# B&R Automation Studio project PROJEKT_AS_4_11_2_75_X20CP1382
Automation Studio 4.9

## Configuration Config1

CPU X20CP1382, AutomationRuntime D4.83, Build 4.1.2, Vc V4.72.3

### Task classes (Cpu.sw)
```
Cyclic#4:
  Program <- Program.prg
Binaries: udbdef, FWRules, TCData, sysconf, Role, User, iomap, ashwd, asfw, arconfig, ashwac
Libraries: runtime, astime, asieccon
```

### Hardware
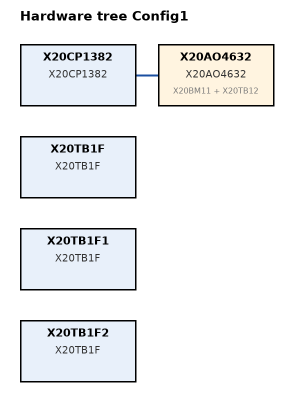
```
X20AO4632 : X20AO4632 v1.2.0.0  [SS1 -> X20TB12.SS; SL -> X20BM11.SL1]
X20BM11 : X20BM11 v1.1.0.0  [X2X1 -> X20CP1382.IF6]
X20CP1382 : X20CP1382 v1.14.0.0  [X1 -> X1.SL; X2 -> X2.SL; X3 -> X3.SL]
  Module X1 (Type=X1, Virtual=true, Version=1.14.0.0)
    Connection (Connector=SS1, TargetModule=X20TB1F, TargetConnector=SS)
    Connection (Connector=SL, TargetModule=X20CP1382, TargetConnector=X1)
  Module X2 (Type=X2, Virtual=true, Version=1.14.0.0)
    Connection (Connector=SS1, TargetModule=X20TB1F1, TargetConnector=SS)
    Connection (Connector=SL, TargetModule=X20CP1382, TargetConnector=X2)
  Module X3 (Type=X3, Virtual=true, Version=1.14.0.0)
    Connection (Connector=SS1, TargetModule=X20TB1F2, TargetConnector=SS)
    Connection (Connector=SL, TargetModule=X20CP1382, TargetConnector=X3)
  Connector IF2:
    ActivateDevice = 1
    Mode = Manual
    InternetAddress = 192.168.10.5
    SubnetMask = 255.255.255.0
    ActivateSnmp = 2
  ConfigurationID = X20CP1382_Config1
  Simulation = 1
X20TB12 : X20TB12 v1.0.0.0
X20TB1F : X20TB1F v1.0.0.0
X20TB1F1 : X20TB1F v1.0.0.0
X20TB1F2 : X20TB1F v1.0.0.0
```

### IoMap.iom - X20CP1382/IoMap.iom
```iecst
VAR_CONFIG
	::Program:speedTreadmill AT %QW."X20AO4632".AnalogOutput01;
	::Program:directionTreadmillright AT %QW."X20AO4632".AnalogOutput02;
	::Program:directionTreadmillleft AT %QW."X20AO4632".AnalogOutput03;
<<<<<<< HEAD
	::Program:Reed_Sensor_Input_1 AT %IW."X1".AnalogInput01;
=======
	::Program:inductiveSensor1_DI AT %IX."X1".DigitalInput01 INVERSE;
	::Program:inductiveSensor2_DI AT %IX."X1".DigitalInput02;
	::Program:peristalticPump1_AO AT %QW."X20AO4632".AnalogOutput04;
>>>>>>> a31492344b22443c312620c2728d9b959337b792
END_VAR
```

## Logical view

### Program Logical/Program

#### Variables.var
```iecst
VAR
	speedTreadmill : INT;
	directionTreadmillleft : INT;
	directionTreadmillright : INT;
<<<<<<< HEAD
	Reed_Sensor_Input_1 : INT;
=======
	inductiveSensor1_DI : BOOL;
	inductiveSensor2_DI : BOOL;
	peristalticPump1_AO : INT;
>>>>>>> a31492344b22443c312620c2728d9b959337b792
END_VAR
```

#### Cyclic.st
```iecst
PROGRAM _CYCLIC
	// IF D11 equals ON -> Power on 10V
	// 32000 = 14,6V
	// 10V =
	speedTreadmill := 30000;
	directionTreadmillleft := 25000;
	//directionTreadmillright := 25000;
	speedTreadmill := -4000;

	peristalticPump1_AO := 10000;
	IF inductiveSensor1_DI = TRUE
	THEN
		directionTreadmillright := 25000;
		directionTreadmillleft := 0;
	ELSIF inductiveSensor2_DI = TRUE THEN
		directionTreadmillleft := 25000;
		directionTreadmillright := 0;
	END_IF;

	//

	//speedTreadmill := -30000;

END_PROGRAM
```

#### Init.st
```iecst
PROGRAM _INIT
	(* Insert code here *)
	currentStation_var := 0;
END_PROGRAM
```
